FUNCTION_BLOCK Step_Motor_Control
VAR_INPUT
END_VAR
VAR_OUTPUT
END_VAR
VAR
END_VAR

// NETWORK 1

END_FUNCTION_BLOCK

(* stored: Version 1.1.0.1, ProductVersion 3.1.4022.7
   POU Step_Motor_Control: Id {5448f867-f1e5-406f-8928-bd3f2f4cae19}, SpecialFunc None *)
